Fanuc KAREL source: kb00186.compact.KL

PROGRAM KB00186
%STACKSIZE=65535
%PRIORITY=65535
%NOLOCKGROUP
VAR
P1 : REAL
RESULT : REAL
BEGIN
P1=1.0
RESULT=SIN(P1)
END KB00186
